// TIA Portal V17 export
// export: Created 2023-12-22T15:04:39.3160294Z, ExportSetting WithDefaults, DisplayName Totally Integrated Automation Portal, DisplayVersion V17, DisplayName TIA Portal Openness, DisplayVersion V17, DisplayName TIA Portal Version Control Interface, DisplayVersion V17, DisplayName STEP 7 Professional, DisplayVersion V17, DisplayName STEP 7 Safety, DisplayVersion V17, DisplayName WinCC Advanced, DisplayVersion V17
ORGANIZATION_BLOCK "Main"   // OB1, LAD, ProgramCycle
TITLE = "Main Program Sweep (Cycle)"
{ S7_Optimized_Access := 'TRUE' }
VERSION : 0.1
// stored: AutoNumber true, IsIECCheckEnabled false, SetENOAutomatically false
   VAR_INPUT
      Initial_Call : Bool;   // Initial call of this OB
      Remanence : Bool;   // =True, if remanent data are available
   END_VAR
   VAR_TEMP   // added for the SCL form of the ladder/FBD networks
      _w1 : Bool;
   END_VAR
BEGIN

REGION Network 1
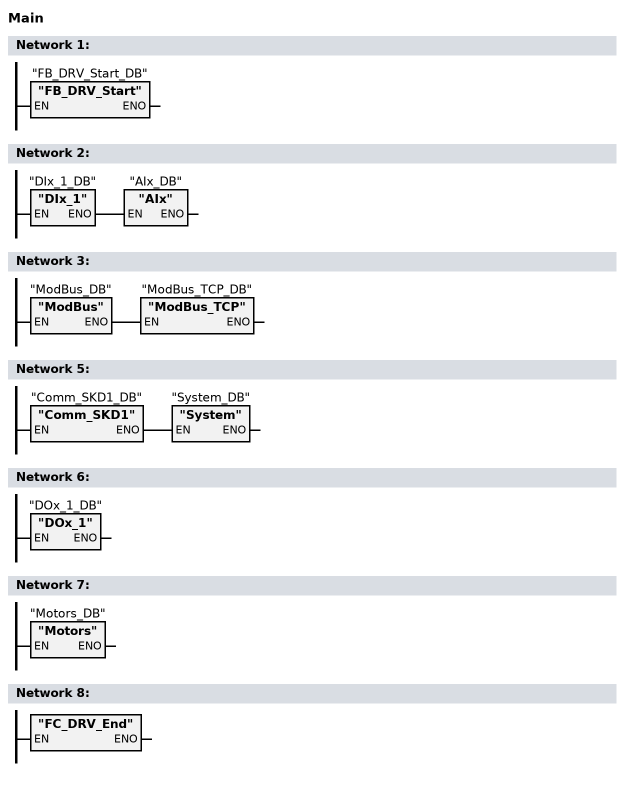
   RUNG wire#powerrail
      "FB_DRV_Start_DB"()
   END_RUNG
   // the same network as SCL:
   "FB_DRV_Start_DB"();   // "FB_DRV_Start"
END_REGION

REGION Network 2
   RUNG wire#powerrail
      "DIx_1_DB"()
      "AIx_DB"()
   END_RUNG
   // the same network as SCL:
   "DIx_1_DB"(ENO => #_w1);   // "DIx_1"
   IF #_w1 THEN
       "AIx_DB"();   // "AIx"
   END_IF;
END_REGION

REGION Network 3
   RUNG wire#powerrail
      "ModBus_DB"()
      "ModBus_TCP_DB"()
   END_RUNG
   // the same network as SCL:
   "ModBus_DB"(ENO => #_w1);   // "ModBus"
   IF #_w1 THEN
       "ModBus_TCP_DB"();   // "ModBus_TCP"
   END_IF;
END_REGION

REGION Network 5
   RUNG wire#powerrail
      "Comm_SKD1_DB"()
      "System_DB"()
   END_RUNG
   // the same network as SCL:
   "Comm_SKD1_DB"(ENO => #_w1);   // "Comm_SKD1"
   IF #_w1 THEN
       "System_DB"();   // "System"
   END_IF;
END_REGION

REGION Network 6
   RUNG wire#powerrail
      "DOx_1_DB"()
   END_RUNG
   // the same network as SCL:
   "DOx_1_DB"();   // "DOx_1"
END_REGION

REGION Network 7
   RUNG wire#powerrail
      "Motors_DB"()
   END_RUNG
   // the same network as SCL:
   "Motors_DB"();   // "Motors"
END_REGION

REGION Network 8
   RUNG wire#powerrail
      "FC_DRV_End"()
   END_RUNG
   // the same network as SCL:
   "FC_DRV_End"();
END_REGION
END_ORGANIZATION_BLOCK
